{attribute 'hide'}
PROGRAM FileSystem_TestSuite
VAR
	nullEntryTest : NullEntry_Test;
	//dirEntryTest : DirectoryEntry_Test;
	//fileEntryTest : FileEntry_Test;
END_VAR

END_PROGRAM

(* stored: Version 1.1.0.1, ProductVersion 3.1.4024.9
   POU FileSystem_TestSuite: Id {2b2ca824-75db-48b8-9b88-c87dc5315cc2}, SpecialFunc None *)
